// TwinCAT 3 PLC project PLCMain
// ProgramVersion: 3.1.4026.12
// CompilerDefines: VISU_USEPROPERTYINFO
// libraries:
//   Tc2_Standard, * (Beckhoff Automation GmbH)
//   Tc2_System, * (Beckhoff Automation GmbH)
//   Tc3_Module, * (Beckhoff Automation GmbH)
// project tree:
//   / GlobalTextList.TcGTLO, PlcTask.TcTTO, Visualization Manager.TcVMO (not stored)
//   POUs/ MAIN.TcPOU, LadderLogicBottleChecker.TcPOU, RecipeManager.TcRMO (not stored)
//   VISUs/ HMI.TcVIS
// real-time tasks:
//   TASK PlcTask: cycle T#10ms, priority 20, ADS port 350
//   TASK PlcTask1: cycle T#10ms, priority 21, ADS port 351

CONFIGURATION PLCMain
    RESOURCE PLC ON TwinCAT3
        TASK PlcTask(INTERVAL := T#10ms, PRIORITY := 21);
        PROGRAM MAIN WITH PlcTask : MAIN;
    END_RESOURCE
END_CONFIGURATION

// ---- POUs/MAIN.TcPOU
PROGRAM MAIN
VAR
END_VAR

LadderLogicBottleChecker();

END_PROGRAM

// ---- POUs/LadderLogicBottleChecker.TcPOU
PROGRAM LadderLogicBottleChecker
VAR
	{attribute 'OPC.UA.DA' := '1'}
	ProximitySensor: BOOL;
	{attribute 'OPC.UA.DA' := '1'}
	BottleDetected: BOOL;
	ProximityTimer: TON;
	{attribute 'OPC.UA.DA' := '1'}
	EjectBottle: BOOL;
	{attribute 'OPC.UA.DA' := '1'}
	EjectRelay: BOOL;
	EjectionTimer: TON;
	{attribute 'OPC.UA.DA' := '1'}
	ExitScript: BOOL;
	
	SessionCounter: CTU;
	{attribute 'OPC.UA.DA' := '1'}
	sessionNumber: INT;
	RejectFlag: BOOL;
	AcceptFlag: BOOL;
END_VAR
VAR // added by the converter: edge detectors and wires of the graphical bodies
    _rt1 : R_TRIG;
END_VAR

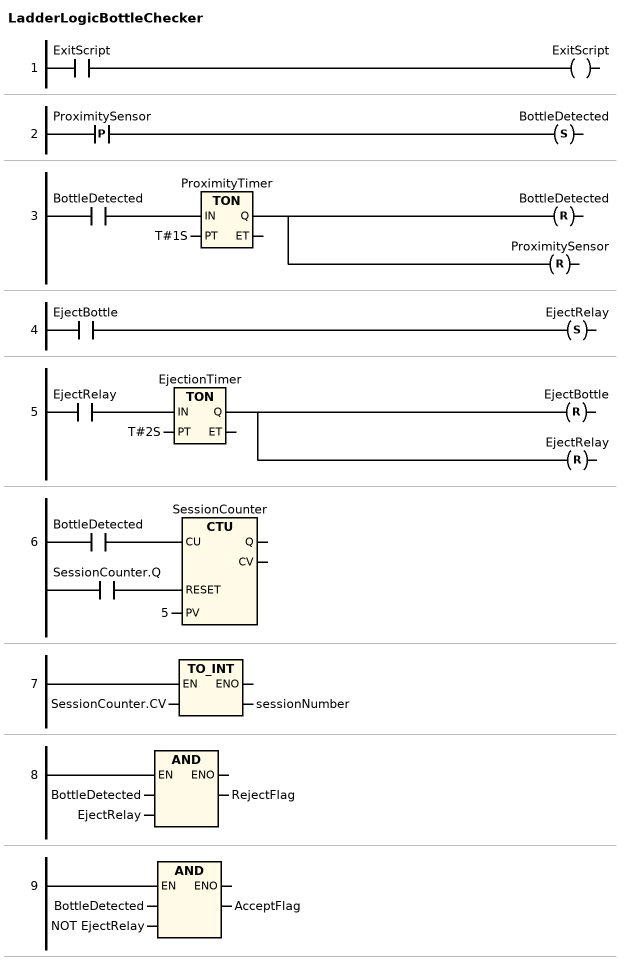
// NETWORK 1
ExitScript := ExitScript;

// NETWORK 2
_rt1(CLK := ProximitySensor);
BottleDetected S= _rt1.Q;

// NETWORK 3
ProximityTimer(IN := BottleDetected, PT := T#1S); // TON
BottleDetected R= ProximityTimer.Q;
ProximitySensor R= ProximityTimer.Q;

// NETWORK 4
EjectRelay S= EjectBottle;

// NETWORK 5
EjectionTimer(IN := EjectRelay, PT := T#2S); // TON
EjectBottle R= EjectionTimer.Q;
EjectRelay R= EjectionTimer.Q;

// NETWORK 6
SessionCounter(CU := BottleDetected, RESET := SessionCounter.Q, PV := 5); // CTU

// NETWORK 7
sessionNumber := TO_INT(SessionCounter.CV);

// NETWORK 8
RejectFlag := BottleDetected AND EjectRelay;

// NETWORK 9
AcceptFlag := BottleDetected AND (NOT EjectRelay);

END_PROGRAM

// ---- GlobalTextList.TcGTLO
TEXTLIST GlobalTextList
  121 = 'Accept'
  8 = 'Eject'
  310 = 'Exit Script'
  56 = 'PrEjectoximity'
  755 = 'Proximity'
  499 = 'Reject'
  589 = 'Start'
  896 = 'Start Script'
  221 = 'Startdef exitScript():\n    return client.get_node("ns=4;s=LadderLogicBottleChecker.ExitScript").get_value()\n'
END_TEXTLIST

// ---- VISUs/HMI.TcVIS
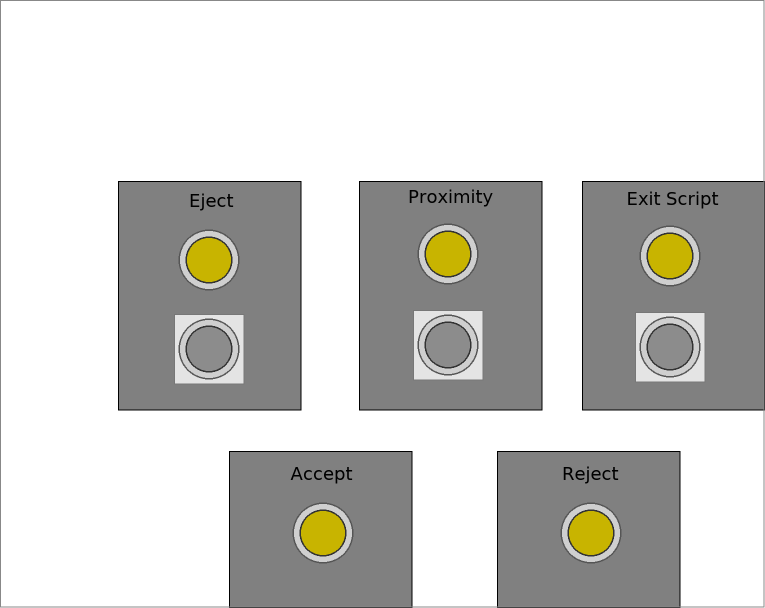
VISUALIZATION HMI  // 765x608
    RoundedRectangle (359,181 183x229)
    PushSwitch (413,310 70x70), variable: LadderLogicBottleChecker.ProximitySensor, behaviour: TOGGLE, style: Switch-PushSwitch-Gray
    Lamp1 (413,219 70x70), variable: LadderLogicBottleChecker.ProximitySensor, style: Lamp-Lamp1-Yellow
    Rectangle (376,183 149x28), "Proximity"
    RoundedRectangle (582,181 183x229)
    PushSwitch (635,312 70x70), variable: LadderLogicBottleChecker.ExitScript, behaviour: TOGGLE, style: Switch-PushSwitch-Gray
    Lamp1 (635,221 70x70), variable: LadderLogicBottleChecker.ExitScript, style: Lamp-Lamp1-Yellow
    Rectangle (598,185 149x28), "Exit Script"
    RoundedRectangle (118,181 183x229)
    PushSwitch (174,314 70x70), variable: LadderLogicBottleChecker.EjectBottle, behaviour: TOGGLE, style: Switch-PushSwitch-Gray
    Lamp1 (174,225 70x70), variable: LadderLogicBottleChecker.EjectRelay, style: Lamp-Lamp1-Yellow
    Rectangle (137,187 149x28), "Eject"
    RoundedRectangle (229,451 183x157)
    Rectangle (247,460 149x28), "Accept"
    RoundedRectangle (497,451 183x157)
    Rectangle (516,460 149x28), "Reject"
    Lamp1 (556,498 70x70), variable: LadderLogicBottleChecker.RejectFlag, style: Lamp-Lamp1-Yellow
    Lamp1 (288,498 70x70), variable: LadderLogicBottleChecker.AcceptFlag, style: Lamp-Lamp1-Yellow
END_VISUALIZATION
